// TIA Portal project "Assembler-Analog" (V15.1)

(* hardware
DEVICE "S7-1200 station_1"  S7-1200 Station
   slot 0: "Rack_0"  S7-1200 Rack  Rack  V1.0
   slot 1: "PLC_1"  CPU 1211C DC/DC/DC  6ES7 211-1AE40-0XB0  V4.2
DEVICE "HMI_1"  KTP900 Basic PN
   slot 0: "HMI_1"  KTP900 Basic PN  6AV2 123-2JB03-0AX0  15.1.0.0
   slot 1: "HMI_RT_1"  KTP900 Basic PN  6AV2 123-2JB03-0AX0  15.1.0.0
   slot 5: "HMI_1.IE_CP_1"  PROFINET Interface  15.0.1.0
      slot 1: "PROFINET Interface_1"  PROFINET Interface
         slot 1: "Port_1"  Port
*)

// ===== PLC "PLC_1"  CPU 1211C DC/DC/DC =====

VAR_GLOBAL   // PLC tag table "Default tag table"
   "Clock_Byte" AT %MB1869 : Byte;
   "Clock_10Hz" AT %M1869.0 : Bool;
   "Clock_5Hz" AT %M1869.1 : Bool;
   "Clock_2.5Hz" AT %M1869.2 : Bool;
   "Clock_2Hz" AT %M1869.3 : Bool;
   "Clock_1.25Hz" AT %M1869.4 : Bool;
   "Clock_1Hz" AT %M1869.5 : Bool;
   "Clock_0.625Hz" AT %M1869.6 : Bool;
   "Clock_0.5Hz" AT %M1869.7 : Bool;
   "System_Byte" AT %MB869 : Byte;
   "FirstScan" AT %M869.0 : Bool;
   "DiagStatusUpdate" AT %M869.1 : Bool;
   "AlwaysTRUE" AT %M869.2 : Bool;
   "AlwaysFALSE" AT %M869.3 : Bool;
END_VAR

VAR_GLOBAL   // PLC tag table "aux"
   "counting_step_1" AT %MW50 : Int;
   "6_box_set_count" AT %MW52 : Int;
   "counting_step_2" AT %MW54 : Int;
   "6_box_set_2" AT %MW56 : Int;
   "pallet_entry_bit" AT %M1.0 : Bool;
   "pallet_fed_entry_bit" AT %M0.6 : Bool;
   "pallet_loaded_bit" AT %M1.3 : Bool;
   "box_2_check_bit" AT %M0.4 : Bool;
   "box_1_check_bit" AT %M0.2 : Bool;
   "turn_cycle_on" AT %M0.3 : Bool;
   "push_limit_bit" AT %M0.5 : Bool;
   "plate_limit_bit" AT %M1.1 : Bool;
   "elevator_moving_bit" AT %M1.2 : Bool;
   "pallet_exit_bit" AT %M1.4 : Bool;
   "tag_1" AT %M1.5 : Bool;
   "tag_2" AT %M1.6 : Bool;
   "tag_3" AT %M1.7 : Bool;
   "tag_4" AT %M2.0 : Bool;
   "tag_5" AT %M2.1 : Bool;
   "box_counting_bit" AT %M0.1 : Bool;
   "2_Box_cycle_complete" AT %M0.0 : Bool;
END_VAR

VAR_GLOBAL   // PLC tag table "I/O_factory"
   "pallet_at_entry" AT %I1.7 : Bool;
   "pallet_at_exit" AT %I2.0 : Bool;
   "pallet_loaded" AT %I2.1 : Bool;
   "box_at_entry" AT %I2.2 : Bool;
   "pusher_limit" AT %I2.3 : Bool;
   "plate_limit" AT %I2.4 : Bool;
   "clamped" AT %I2.5 : Bool;
   "elevator_moving" AT %I2.6 : Bool;
   "start" AT %I1.0 : Bool;
   "reset" AT %I1.1 : Bool;
   "stop" AT %I1.2 : Bool;
   "emergency_stop" AT %I1.3 : Bool;
   "auto" AT %I1.4 : Bool;
   "running" AT %I1.5 : Bool;
   "pallet_feeder" AT %Q0.0 : Bool;
   "load_pallet" AT %Q0.1 : Bool;
   "exit_conveyor" AT %Q0.2 : Bool;
   "move_to_limit" AT %Q0.3 : Bool;
   "elevator_up" AT %Q0.4 : Bool;
   "elevator_down" AT %Q0.5 : Bool;
   "box_feeder" AT %Q0.6 : Bool;
   "turn" AT %Q0.7 : Bool;
   "push" AT %Q1.0 : Bool;
   "load_belt" AT %Q1.1 : Bool;
   "clamp" AT %Q1.2 : Bool;
   "open_plate" AT %Q1.3 : Bool;
   "warning_light" AT %Q1.4 : Bool;
   "start_light" AT %Q1.5 : Bool;
   "reset_light" AT %Q1.6 : Bool;
   "stop_light" AT %Q1.7 : Bool;
   "counter" AT %QD30 : DInt;
   "manual" AT %I1.6 : Bool;
END_VAR

DATA_BLOCK "Auxiliare"   // DB1
{ S7_Optimized_Access := 'TRUE' }
VERSION : 0.1
   VAR
      step_counter_1 : Int;
      "6_box_set_count_1" : Int;
      step_count_2 : Int;
      "6_box_set_count_2" : Int;
      "counter" : Int;
      "mod" : DInt;
      turn_cycle_on : Bool;
      system_stop : Bool;
      pallet_entry_elevbit : Bool;
      pallet_fed_entry_bit : Bool;
      pallet_loaded_bit : Bool;
      box2_check_bit : Bool;
      box1_check_bit : Bool;
      "2_box_cycle_complete" : Bool;
      pusher_limit_bit : Bool;
      plate_limit_bit : Bool;
      elevator_moving_bit : Bool;
      pallet_exit_bit : Bool;
      aux1 : Bool;
      aux2 : Bool;
      aux3 : Bool;
      aux4 : Bool;
      aux5 : Bool;
      box_counting_bit : Bool;
   END_VAR
BEGIN
END_DATA_BLOCK

// folder: FBs/Cutii

DATA_BLOCK "Cutii_FB_DB"   // DB5
{ S7_Optimized_Access := 'TRUE' }
VERSION : 0.1
// stored: InstanceOfName Cutii_FB
"Cutii_FB"
BEGIN
END_DATA_BLOCK

// folder: FBs/Paleti

DATA_BLOCK "Paleti_FB_DB"   // DB4
{ S7_Optimized_Access := 'TRUE' }
VERSION : 0.1
// stored: InstanceOfName Paleti_FB
"Paleti_FB"
BEGIN
END_DATA_BLOCK

// folder: FBs/Paletizor

DATA_BLOCK "Paletizor_FB_DB"   // DB2
{ S7_Optimized_Access := 'TRUE' }
VERSION : 0.1
// stored: InstanceOfName Paletizor_FB
"Paletizor_FB"
BEGIN
END_DATA_BLOCK

// folder: System blocks/Program resources

DATA_BLOCK "2_box_timer"   // DB3
{ S7_Optimized_Access := 'TRUE' }
AUTHOR : Simatic
FAMILY : IEC
NAME : IEC_TMR
VERSION : 1.0
// stored: InstanceOfName IEC_TIMER
"IEC_TIMER"
BEGIN
END_DATA_BLOCK

DATA_BLOCK "3_box_timer"   // DB7
{ S7_Optimized_Access := 'TRUE' }
AUTHOR : Simatic
FAMILY : IEC
NAME : IEC_TMR
VERSION : 1.0
// stored: InstanceOfName IEC_TIMER
"IEC_TIMER"
BEGIN
END_DATA_BLOCK

// folder: (top level)

FUNCTION "paletizor" : Void   // FC1, LAD
{ S7_Optimized_Access := 'TRUE' }
VERSION : 0.1
   VAR_TEMP   // added for the SCL form of the ladder/FBD networks
      _w1 : Bool;
      _w2 : Bool;
      _w3 : Bool;
   END_VAR
BEGIN

REGION Network 1: butoane start, stop, reset si esd
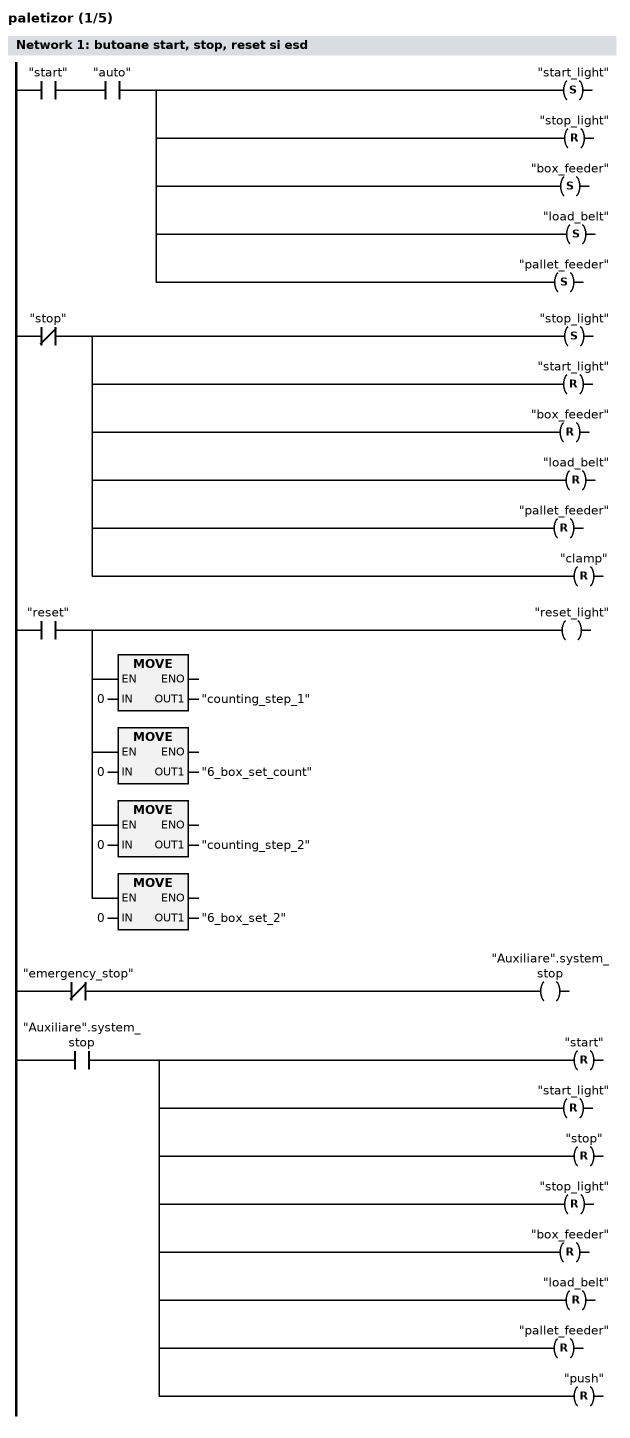
   RUNG wire#powerrail
      Contact( "start" )
      Contact( "auto" )
      wire#w1
      S_Coil( "start_light" )
   END_RUNG
   RUNG wire#w1
      R_Coil( "stop_light" )
   END_RUNG
   RUNG wire#w1
      S_Coil( "box_feeder" )
   END_RUNG
   RUNG wire#w1
      S_Coil( "load_belt" )
   END_RUNG
   RUNG wire#w1
      S_Coil( "pallet_feeder" )
   END_RUNG
   RUNG wire#powerrail
      I_Contact( "stop" )
      wire#w2
      S_Coil( "stop_light" )
   END_RUNG
   RUNG wire#w2
      R_Coil( "start_light" )
   END_RUNG
   RUNG wire#w2
      R_Coil( "box_feeder" )
   END_RUNG
   RUNG wire#w2
      R_Coil( "load_belt" )
   END_RUNG
   RUNG wire#w2
      R_Coil( "pallet_feeder" )
   END_RUNG
   RUNG wire#w2
      R_Coil( "clamp" )
   END_RUNG
   RUNG wire#powerrail
      Contact( "reset" )
      wire#w3
      Coil( "reset_light" )
   END_RUNG
   RUNG wire#w3
      Move(in := 0, out1 => "counting_step_1")
   END_RUNG
   RUNG wire#w3
      Move(in := 0, out1 => "6_box_set_count")
   END_RUNG
   RUNG wire#w3
      Move(in := 0, out1 => "counting_step_2")
   END_RUNG
   RUNG wire#w3
      Move(in := 0, out1 => "6_box_set_2")
   END_RUNG
   RUNG wire#powerrail
      I_Contact( "emergency_stop" )
      Coil( "Auxiliare".system_stop )
   END_RUNG
   RUNG wire#powerrail
      Contact( "Auxiliare".system_stop )
      wire#w4
      R_Coil( "start" )
   END_RUNG
   RUNG wire#w4
      R_Coil( "start_light" )
   END_RUNG
   RUNG wire#w4
      R_Coil( "stop" )
   END_RUNG
   RUNG wire#w4
      R_Coil( "stop_light" )
   END_RUNG
   RUNG wire#w4
      R_Coil( "box_feeder" )
   END_RUNG
   RUNG wire#w4
      R_Coil( "load_belt" )
   END_RUNG
   RUNG wire#w4
      R_Coil( "pallet_feeder" )
   END_RUNG
   RUNG wire#w4
      R_Coil( "push" )
   END_RUNG
   // the same network as SCL:
   IF "start" AND "auto" THEN
       "start_light" := TRUE;
       "stop_light" := FALSE;
       "box_feeder" := TRUE;
       "load_belt" := TRUE;
       "pallet_feeder" := TRUE;
   END_IF;
   IF NOT "stop" THEN
       "stop_light" := TRUE;
       "start_light" := FALSE;
       "box_feeder" := FALSE;
       "load_belt" := FALSE;
       "pallet_feeder" := FALSE;
       "clamp" := FALSE;
   END_IF;
   "reset_light" := "reset";
   IF "reset" THEN
       "counting_step_1" := 0;
       "6_box_set_count" := 0;
       "counting_step_2" := 0;
       "6_box_set_2" := 0;
   END_IF;
   "Auxiliare".system_stop := NOT "emergency_stop";
   IF "Auxiliare".system_stop THEN
       "start" := FALSE;
       "start_light" := FALSE;
       "stop" := FALSE;
       "stop_light" := FALSE;
       "box_feeder" := FALSE;
       "load_belt" := FALSE;
       "pallet_feeder" := FALSE;
       "push" := FALSE;
   END_IF;
END_REGION

REGION Network 2: palet la intrare
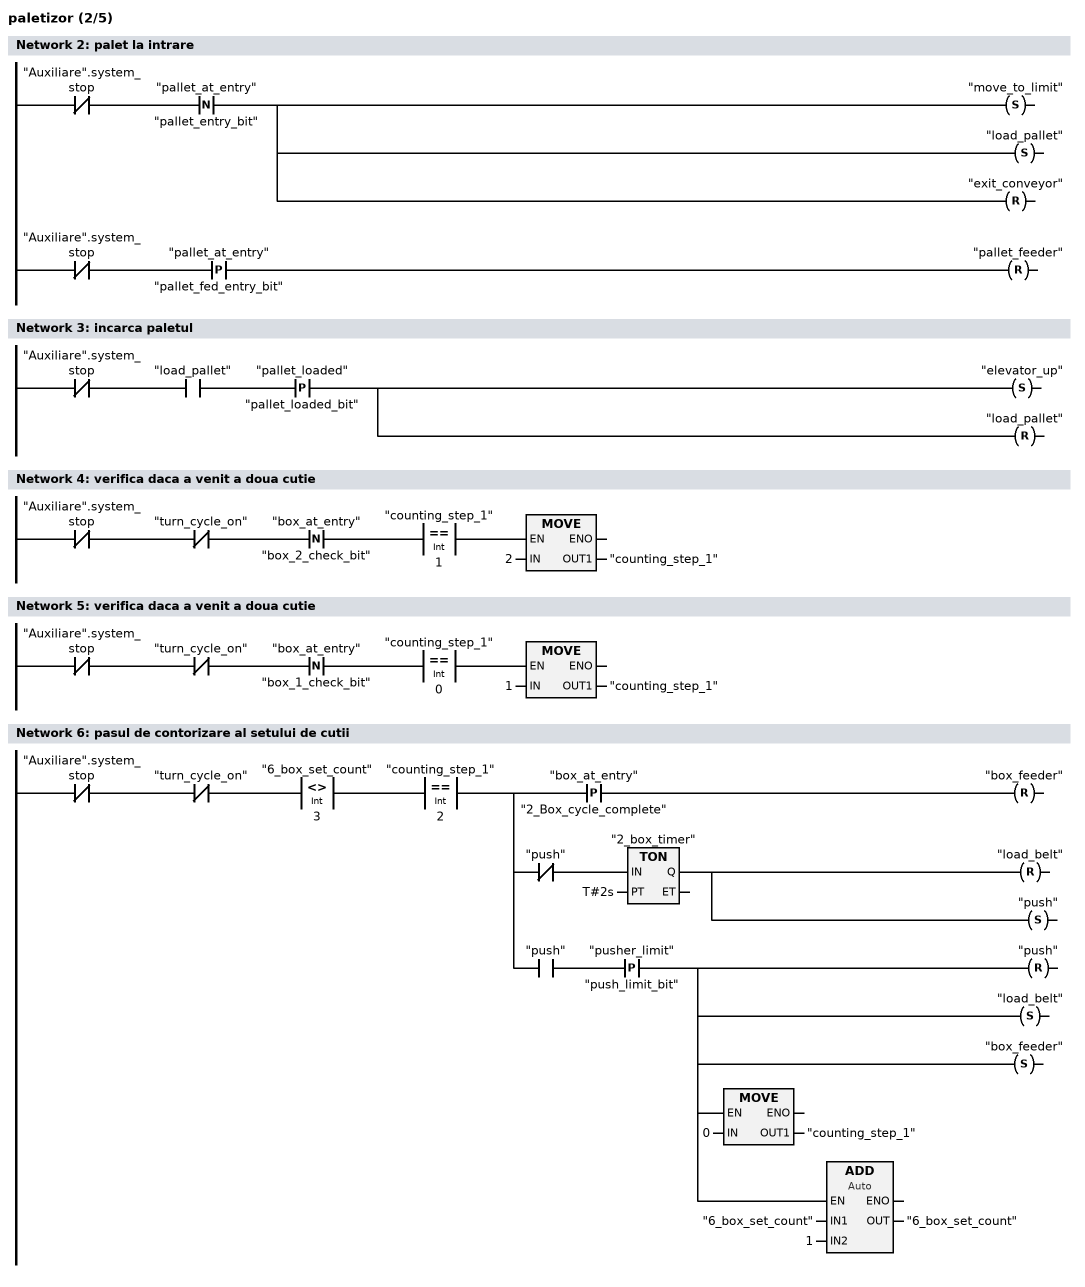
   RUNG wire#powerrail
      I_Contact( "Auxiliare".system_stop )
      N_Contact(operand := "pallet_at_entry", bit := "pallet_entry_bit")
      wire#w1
      S_Coil( "move_to_limit" )
   END_RUNG
   RUNG wire#w1
      S_Coil( "load_pallet" )
   END_RUNG
   RUNG wire#w1
      R_Coil( "exit_conveyor" )
   END_RUNG
   RUNG wire#powerrail
      I_Contact( "Auxiliare".system_stop )
      P_Contact(operand := "pallet_at_entry", bit := "pallet_fed_entry_bit")
      R_Coil( "pallet_feeder" )
   END_RUNG
   // the same network as SCL:
   #_w1 := NOT "Auxiliare".system_stop AND NOT "pallet_at_entry" AND "pallet_entry_bit";   // falling edge of "pallet_at_entry"
   "pallet_entry_bit" := "pallet_at_entry";
   IF #_w1 THEN
       "move_to_limit" := TRUE;
       "load_pallet" := TRUE;
       "exit_conveyor" := FALSE;
   END_IF;
   #_w2 := NOT "Auxiliare".system_stop AND "pallet_at_entry" AND NOT "pallet_fed_entry_bit";   // rising edge of "pallet_at_entry"
   "pallet_fed_entry_bit" := "pallet_at_entry";
   IF #_w2 THEN "pallet_feeder" := FALSE; END_IF;
END_REGION

REGION Network 3: incarca paletul
   RUNG wire#powerrail
      I_Contact( "Auxiliare".system_stop )
      Contact( "load_pallet" )
      P_Contact(operand := "pallet_loaded", bit := "pallet_loaded_bit")
      wire#w1
      S_Coil( "elevator_up" )
   END_RUNG
   RUNG wire#w1
      R_Coil( "load_pallet" )
   END_RUNG
   // the same network as SCL:
   #_w1 := NOT "Auxiliare".system_stop AND "load_pallet" AND "pallet_loaded" AND NOT "pallet_loaded_bit";   // rising edge of "pallet_loaded"
   "pallet_loaded_bit" := "pallet_loaded";
   IF #_w1 THEN
       "elevator_up" := TRUE;
       "load_pallet" := FALSE;
   END_IF;
END_REGION

REGION Network 4: verifica daca a venit a doua cutie
   RUNG wire#powerrail
      I_Contact( "Auxiliare".system_stop )
      I_Contact( "turn_cycle_on" )
      N_Contact(operand := "box_at_entry", bit := "box_2_check_bit")
      { S7_Templates := "SrcType := Int" } EQ_Contact(in1 := "counting_step_1", in2 := 1)
      Move(in := 2, out1 => "counting_step_1")
   END_RUNG
   // the same network as SCL:
   #_w1 := NOT "Auxiliare".system_stop AND NOT "turn_cycle_on" AND NOT "box_at_entry" AND "box_2_check_bit";   // falling edge of "box_at_entry"
   "box_2_check_bit" := "box_at_entry";
   IF #_w1 AND ("counting_step_1" = 1) THEN "counting_step_1" := 2; END_IF;
END_REGION

REGION Network 5: verifica daca a venit a doua cutie
   RUNG wire#powerrail
      I_Contact( "Auxiliare".system_stop )
      I_Contact( "turn_cycle_on" )
      N_Contact(operand := "box_at_entry", bit := "box_1_check_bit")
      { S7_Templates := "SrcType := Int" } EQ_Contact(in1 := "counting_step_1", in2 := 0)
      Move(in := 1, out1 => "counting_step_1")
   END_RUNG
   // the same network as SCL:
   #_w1 := NOT "Auxiliare".system_stop AND NOT "turn_cycle_on" AND NOT "box_at_entry" AND "box_1_check_bit";   // falling edge of "box_at_entry"
   "box_1_check_bit" := "box_at_entry";
   IF #_w1 AND ("counting_step_1" = 0) THEN "counting_step_1" := 1; END_IF;
END_REGION

REGION Network 6: pasul de contorizare al setului de cutii
   #_w1 := NOT "Auxiliare".system_stop AND NOT "turn_cycle_on" AND ("6_box_set_count" <> 3) AND ("counting_step_1" = 2);
   #_w2 := #_w1 AND "box_at_entry" AND NOT "2_Box_cycle_complete";   // rising edge of "box_at_entry"
   "2_Box_cycle_complete" := "box_at_entry";
   IF #_w2 THEN "box_feeder" := FALSE; END_IF;
   "2_box_timer".TON(IN := #_w1 AND NOT "push", PT := T#2s);
   IF "2_box_timer".Q THEN
       "load_belt" := FALSE;
       "push" := TRUE;
   END_IF;
   #_w3 := #_w1 AND "push" AND "pusher_limit" AND NOT "push_limit_bit";   // rising edge of "pusher_limit"
   "push_limit_bit" := "pusher_limit";
   IF #_w3 THEN
       "push" := FALSE;
       "load_belt" := TRUE;
       "box_feeder" := TRUE;
       "counting_step_1" := 0;
       "6_box_set_count" := "6_box_set_count" + 1;
   END_IF;
END_REGION

REGION Network 7: daca s a format setul, sa dea clamp
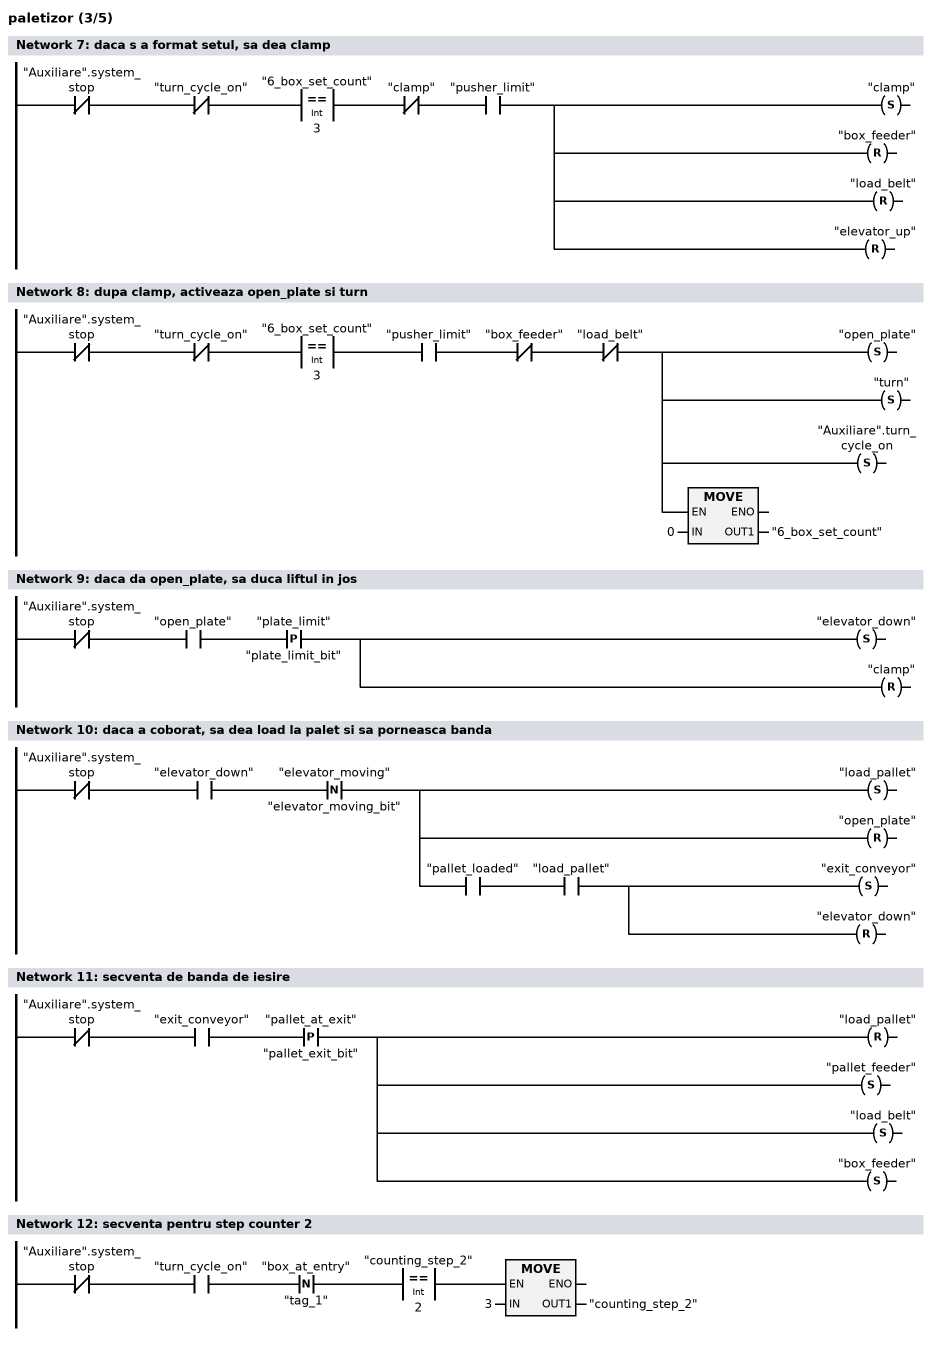
   RUNG wire#powerrail
      I_Contact( "Auxiliare".system_stop )
      I_Contact( "turn_cycle_on" )
      { S7_Templates := "SrcType := Int" } EQ_Contact(in1 := "6_box_set_count", in2 := 3)
      I_Contact( "clamp" )
      Contact( "pusher_limit" )
      wire#w1
      S_Coil( "clamp" )
   END_RUNG
   RUNG wire#w1
      R_Coil( "box_feeder" )
   END_RUNG
   RUNG wire#w1
      R_Coil( "load_belt" )
   END_RUNG
   RUNG wire#w1
      R_Coil( "elevator_up" )
   END_RUNG
   // the same network as SCL:
   #_w1 := NOT "Auxiliare".system_stop AND NOT "turn_cycle_on" AND ("6_box_set_count" = 3) AND NOT "clamp" AND "pusher_limit";
   IF #_w1 THEN
       "clamp" := TRUE;
       "box_feeder" := FALSE;
       "load_belt" := FALSE;
       "elevator_up" := FALSE;
   END_IF;
END_REGION

REGION Network 8: dupa clamp, activeaza open_plate si turn
   RUNG wire#powerrail
      I_Contact( "Auxiliare".system_stop )
      I_Contact( "turn_cycle_on" )
      { S7_Templates := "SrcType := Int" } EQ_Contact(in1 := "6_box_set_count", in2 := 3)
      Contact( "pusher_limit" )
      I_Contact( "box_feeder" )
      I_Contact( "load_belt" )
      wire#w1
      S_Coil( "open_plate" )
   END_RUNG
   RUNG wire#w1
      S_Coil( "turn" )
   END_RUNG
   RUNG wire#w1
      S_Coil( "Auxiliare".turn_cycle_on )
   END_RUNG
   RUNG wire#w1
      Move(in := 0, out1 => "6_box_set_count")
   END_RUNG
   // the same network as SCL:
   IF NOT "Auxiliare".system_stop AND NOT "turn_cycle_on" AND ("6_box_set_count" = 3) AND "pusher_limit" AND NOT "box_feeder" AND NOT "load_belt" THEN
       "open_plate" := TRUE;
       "turn" := TRUE;
       "Auxiliare".turn_cycle_on := TRUE;
       "6_box_set_count" := 0;
   END_IF;
END_REGION

REGION Network 9: daca da open_plate, sa duca liftul in jos
   RUNG wire#powerrail
      I_Contact( "Auxiliare".system_stop )
      Contact( "open_plate" )
      P_Contact(operand := "plate_limit", bit := "plate_limit_bit")
      wire#w1
      S_Coil( "elevator_down" )
   END_RUNG
   RUNG wire#w1
      R_Coil( "clamp" )
   END_RUNG
   // the same network as SCL:
   #_w1 := NOT "Auxiliare".system_stop AND "open_plate" AND "plate_limit" AND NOT "plate_limit_bit";   // rising edge of "plate_limit"
   "plate_limit_bit" := "plate_limit";
   IF #_w1 THEN
       "elevator_down" := TRUE;
       "clamp" := FALSE;
   END_IF;
END_REGION

REGION Network 10: daca a coborat, sa dea load la palet si sa porneasca banda
   RUNG wire#powerrail
      I_Contact( "Auxiliare".system_stop )
      Contact( "elevator_down" )
      N_Contact(operand := "elevator_moving", bit := "elevator_moving_bit")
      wire#w1
      S_Coil( "load_pallet" )
   END_RUNG
   RUNG wire#w1
      R_Coil( "open_plate" )
   END_RUNG
   RUNG wire#w1
      Contact( "pallet_loaded" )
      Contact( "load_pallet" )
      wire#w2
      S_Coil( "exit_conveyor" )
   END_RUNG
   RUNG wire#w2
      R_Coil( "elevator_down" )
   END_RUNG
   // the same network as SCL:
   #_w1 := NOT "Auxiliare".system_stop AND "elevator_down" AND NOT "elevator_moving" AND "elevator_moving_bit";   // falling edge of "elevator_moving"
   "elevator_moving_bit" := "elevator_moving";
   IF #_w1 THEN
       "load_pallet" := TRUE;
       "open_plate" := FALSE;
   END_IF;
   IF #_w1 AND "pallet_loaded" AND "load_pallet" THEN
       "exit_conveyor" := TRUE;
       "elevator_down" := FALSE;
   END_IF;
END_REGION

REGION Network 11: secventa de banda de iesire
   RUNG wire#powerrail
      I_Contact( "Auxiliare".system_stop )
      Contact( "exit_conveyor" )
      P_Contact(operand := "pallet_at_exit", bit := "pallet_exit_bit")
      wire#w1
      R_Coil( "load_pallet" )
   END_RUNG
   RUNG wire#w1
      S_Coil( "pallet_feeder" )
   END_RUNG
   RUNG wire#w1
      S_Coil( "load_belt" )
   END_RUNG
   RUNG wire#w1
      S_Coil( "box_feeder" )
   END_RUNG
   // the same network as SCL:
   #_w1 := NOT "Auxiliare".system_stop AND "exit_conveyor" AND "pallet_at_exit" AND NOT "pallet_exit_bit";   // rising edge of "pallet_at_exit"
   "pallet_exit_bit" := "pallet_at_exit";
   IF #_w1 THEN
       "load_pallet" := FALSE;
       "pallet_feeder" := TRUE;
       "load_belt" := TRUE;
       "box_feeder" := TRUE;
   END_IF;
END_REGION

REGION Network 12: secventa pentru step counter 2
   RUNG wire#powerrail
      I_Contact( "Auxiliare".system_stop )
      Contact( "turn_cycle_on" )
      N_Contact(operand := "box_at_entry", bit := "tag_1")
      { S7_Templates := "SrcType := Int" } EQ_Contact(in1 := "counting_step_2", in2 := 2)
      Move(in := 3, out1 => "counting_step_2")
   END_RUNG
   // the same network as SCL:
   #_w1 := NOT "Auxiliare".system_stop AND "turn_cycle_on" AND NOT "box_at_entry" AND "tag_1";   // falling edge of "box_at_entry"
   "tag_1" := "box_at_entry";
   IF #_w1 AND ("counting_step_2" = 2) THEN "counting_step_2" := 3; END_IF;
END_REGION

REGION Network 13: secventa pentru step counter 2, partea precedenta
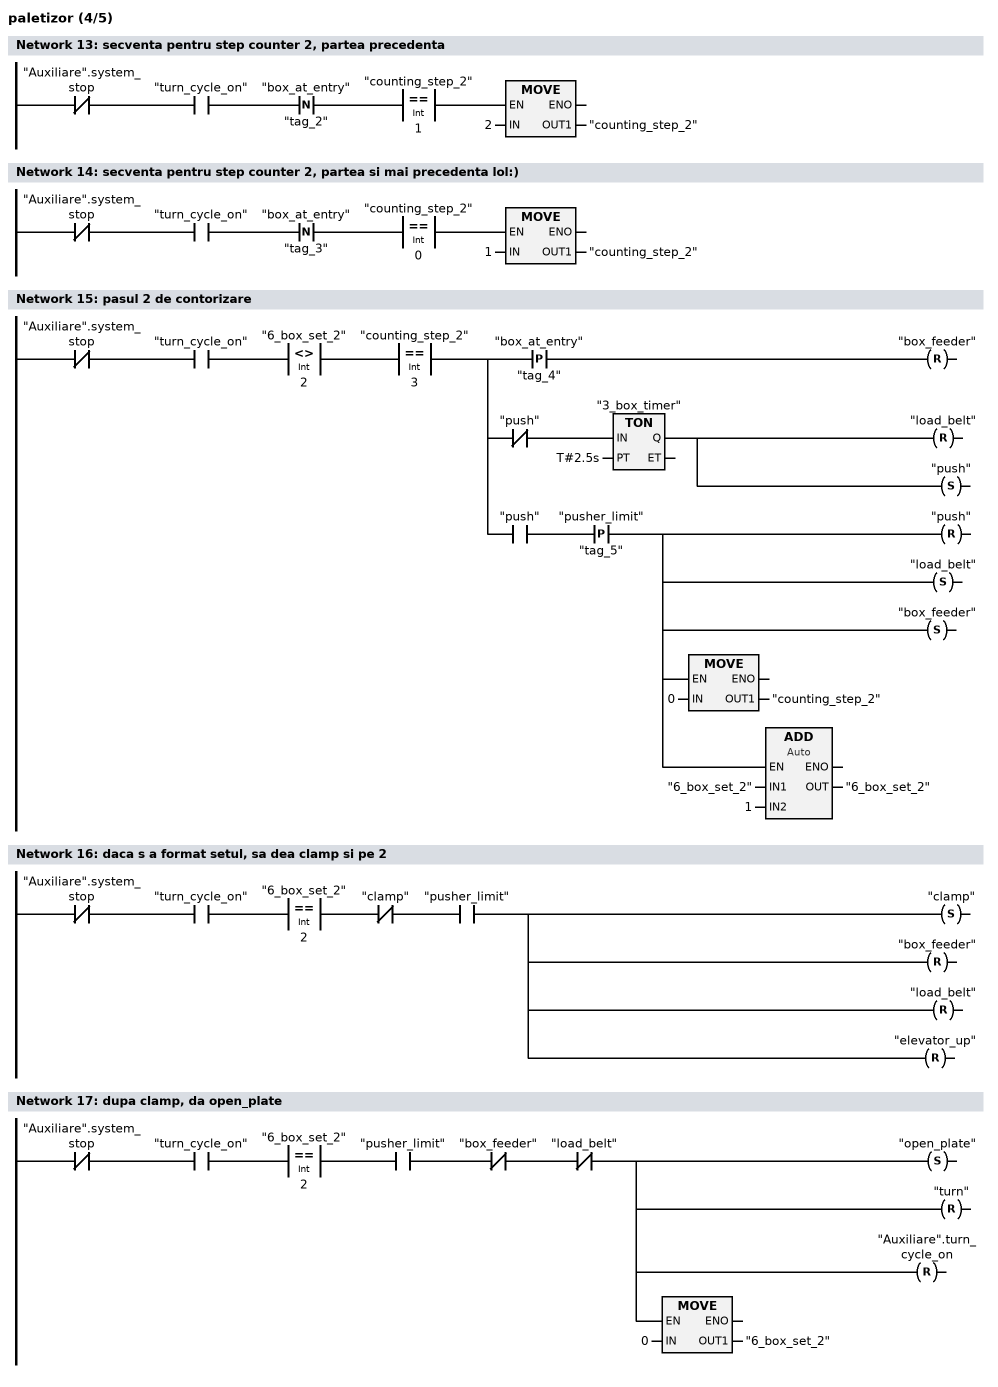
   RUNG wire#powerrail
      I_Contact( "Auxiliare".system_stop )
      Contact( "turn_cycle_on" )
      N_Contact(operand := "box_at_entry", bit := "tag_2")
      { S7_Templates := "SrcType := Int" } EQ_Contact(in1 := "counting_step_2", in2 := 1)
      Move(in := 2, out1 => "counting_step_2")
   END_RUNG
   // the same network as SCL:
   #_w1 := NOT "Auxiliare".system_stop AND "turn_cycle_on" AND NOT "box_at_entry" AND "tag_2";   // falling edge of "box_at_entry"
   "tag_2" := "box_at_entry";
   IF #_w1 AND ("counting_step_2" = 1) THEN "counting_step_2" := 2; END_IF;
END_REGION

REGION Network 14: secventa pentru step counter 2, partea si mai precedenta lol:)
   RUNG wire#powerrail
      I_Contact( "Auxiliare".system_stop )
      Contact( "turn_cycle_on" )
      N_Contact(operand := "box_at_entry", bit := "tag_3")
      { S7_Templates := "SrcType := Int" } EQ_Contact(in1 := "counting_step_2", in2 := 0)
      Move(in := 1, out1 => "counting_step_2")
   END_RUNG
   // the same network as SCL:
   #_w1 := NOT "Auxiliare".system_stop AND "turn_cycle_on" AND NOT "box_at_entry" AND "tag_3";   // falling edge of "box_at_entry"
   "tag_3" := "box_at_entry";
   IF #_w1 AND ("counting_step_2" = 0) THEN "counting_step_2" := 1; END_IF;
END_REGION

REGION Network 15: pasul 2 de contorizare
   #_w1 := NOT "Auxiliare".system_stop AND "turn_cycle_on" AND ("6_box_set_2" <> 2) AND ("counting_step_2" = 3);
   #_w2 := #_w1 AND "box_at_entry" AND NOT "tag_4";   // rising edge of "box_at_entry"
   "tag_4" := "box_at_entry";
   IF #_w2 THEN "box_feeder" := FALSE; END_IF;
   "3_box_timer".TON(IN := #_w1 AND NOT "push", PT := T#2.5s);
   IF "3_box_timer".Q THEN
       "load_belt" := FALSE;
       "push" := TRUE;
   END_IF;
   #_w3 := #_w1 AND "push" AND "pusher_limit" AND NOT "tag_5";   // rising edge of "pusher_limit"
   "tag_5" := "pusher_limit";
   IF #_w3 THEN
       "push" := FALSE;
       "load_belt" := TRUE;
       "box_feeder" := TRUE;
       "counting_step_2" := 0;
       "6_box_set_2" := "6_box_set_2" + 1;
   END_IF;
END_REGION

REGION Network 16: daca s a format setul, sa dea clamp si pe 2
   RUNG wire#powerrail
      I_Contact( "Auxiliare".system_stop )
      Contact( "turn_cycle_on" )
      { S7_Templates := "SrcType := Int" } EQ_Contact(in1 := "6_box_set_2", in2 := 2)
      I_Contact( "clamp" )
      Contact( "pusher_limit" )
      wire#w1
      S_Coil( "clamp" )
   END_RUNG
   RUNG wire#w1
      R_Coil( "box_feeder" )
   END_RUNG
   RUNG wire#w1
      R_Coil( "load_belt" )
   END_RUNG
   RUNG wire#w1
      R_Coil( "elevator_up" )
   END_RUNG
   // the same network as SCL:
   #_w1 := NOT "Auxiliare".system_stop AND "turn_cycle_on" AND ("6_box_set_2" = 2) AND NOT "clamp" AND "pusher_limit";
   IF #_w1 THEN
       "clamp" := TRUE;
       "box_feeder" := FALSE;
       "load_belt" := FALSE;
       "elevator_up" := FALSE;
   END_IF;
END_REGION

REGION Network 17: dupa clamp, da open_plate
   RUNG wire#powerrail
      I_Contact( "Auxiliare".system_stop )
      Contact( "turn_cycle_on" )
      { S7_Templates := "SrcType := Int" } EQ_Contact(in1 := "6_box_set_2", in2 := 2)
      Contact( "pusher_limit" )
      I_Contact( "box_feeder" )
      I_Contact( "load_belt" )
      wire#w1
      S_Coil( "open_plate" )
   END_RUNG
   RUNG wire#w1
      R_Coil( "turn" )
   END_RUNG
   RUNG wire#w1
      R_Coil( "Auxiliare".turn_cycle_on )
   END_RUNG
   RUNG wire#w1
      Move(in := 0, out1 => "6_box_set_2")
   END_RUNG
   // the same network as SCL:
   IF NOT "Auxiliare".system_stop AND "turn_cycle_on" AND ("6_box_set_2" = 2) AND "pusher_limit" AND NOT "box_feeder" AND NOT "load_belt" THEN
       "open_plate" := TRUE;
       "turn" := FALSE;
       "Auxiliare".turn_cycle_on := FALSE;
       "6_box_set_2" := 0;
   END_IF;
END_REGION

REGION Network 18: daca s a terminat, da increment la counter
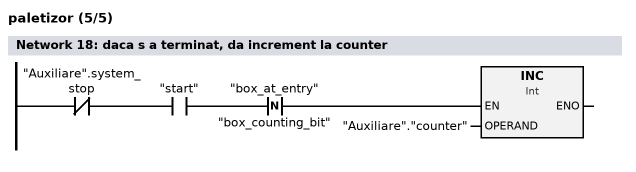
   RUNG wire#powerrail
      I_Contact( "Auxiliare".system_stop )
      Contact( "start" )
      N_Contact(operand := "box_at_entry", bit := "box_counting_bit")
      { S7_Templates := "DestType := Int" } Inc( "Auxiliare"."counter" )
   END_RUNG
   // the same network as SCL:
   #_w1 := NOT "Auxiliare".system_stop AND "start" AND NOT "box_at_entry" AND "box_counting_bit";   // falling edge of "box_at_entry"
   "box_counting_bit" := "box_at_entry";
   IF #_w1 THEN "Auxiliare"."counter" := "Auxiliare"."counter" + 1; END_IF;
END_REGION
END_FUNCTION

FUNCTION "MHJ-PLC-Lab-Function-S71200" : Void   // FC9000, SCL
{ S7_Optimized_Access := 'TRUE' }
VERSION : 0.1
   VAR_TEMP
      rdTimeReturn : Int;
      outputTime : DTL;
      SyncVal : Byte;
      forVal : Int;
      forVal_2 : Int;
      Value : Byte;
   END_VAR
   VAR CONSTANT
      CompVal : Byte := 16#34;
      Value_01 : Byte := 16#11;
      Value_01_DW : DWord := 16#A165_D992;
      Value_02_DW : DWord := 16#58BE_4401;
   END_VAR
BEGIN

   #Value:=PEEK(area := 16#82,
        dbNumber := 0,
        byteOffset := 511);
   #Value := #Value + 1;

   POKE(area := 16#82,
        dbNumber := 0,
        byteOffset := 511,
        value := #Value);

   POKE(area:=16#81,
        dbNumber:=0,
        byteOffset:=1016,
        value:=#Value_01_DW);
   POKE(area := 16#81,
        dbNumber := 0,
        byteOffset := 1020,
        value := #Value_02_DW);

   POKE(area := 16#81,
        dbNumber := 0,
        byteOffset := 511,
        value := B#16#00);

   FOR #forVal := 0 TO 120 DO
       FOR #forVal_2:=0 TO 10 DO
           #rdTimeReturn:=RD_SYS_T(#outputTime);
           #rdTimeReturn := WR_SYS_T(#outputTime);
           #rdTimeReturn := RD_SYS_T(#outputTime);
           #rdTimeReturn := WR_SYS_T(#outputTime);
       END_FOR;
       #SyncVal:= PEEK(area := 16#81,
                      dbNumber := 0,
                      byteOffset := 511);
       IF #SyncVal = #CompVal THEN
          GOTO M_1;
       END_IF;
   END_FOR;
   RETURN;

   M_1:
   POKE(area := 16#81,
        dbNumber := 0,
        byteOffset := 511,
        value := B#16#0);
END_FUNCTION

ORGANIZATION_BLOCK "Main"   // OB1, LAD, ProgramCycle
TITLE = "Main Program Sweep (Cycle)"
{ S7_Optimized_Access := 'TRUE' }
VERSION : 0.1
   VAR_INPUT
      Initial_Call : Bool;   // Initial call of this OB
      Remanence : Bool;   // =True, if remanent data are available
   END_VAR
BEGIN

REGION Network 1: fct de conectare la factory io
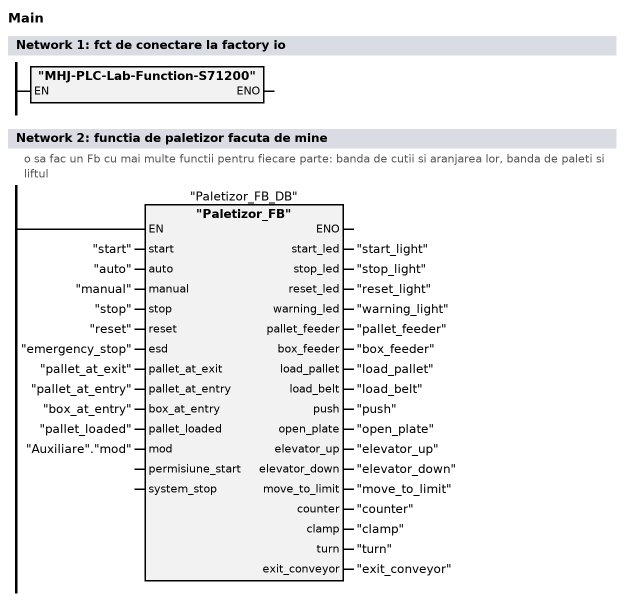
   RUNG wire#powerrail
      "MHJ-PLC-Lab-Function-S71200"()
   END_RUNG
   // the same network as SCL:
   "MHJ-PLC-Lab-Function-S71200"();
END_REGION

REGION Network 2: functia de paletizor facuta de mine
   // o sa fac un Fb cu mai multe functii pentru fiecare parte: banda de cutii si aranjarea lor, banda de paleti si  liftul
   RUNG wire#powerrail
      "Paletizor_FB_DB"(start := "start", auto := "auto", manual := "manual", stop := "stop", reset := "reset", esd := "emergency_stop", pallet_at_exit := "pallet_at_exit", pallet_at_entry := "pallet_at_entry", box_at_entry := "box_at_entry", pallet_loaded := "pallet_loaded", "mod" := "Auxiliare"."mod", permisiune_start :=, system_stop :=, start_led => "start_light", stop_led => "stop_light", reset_led => "reset_light", warning_led => "warning_light", pallet_feeder => "pallet_feeder", box_feeder => "box_feeder", load_pallet => "load_pallet", load_belt => "load_belt", push => "push", open_plate => "open_plate", elevator_up => "elevator_up", elevator_down => "elevator_down", move_to_limit => "move_to_limit", "counter" => "counter", clamp => "clamp", turn => "turn", exit_conveyor => "exit_conveyor")
   END_RUNG
   // the same network as SCL:
   "Paletizor_FB_DB"(start := "start",   // "Paletizor_FB"
                     auto := "auto",
                     manual := "manual",
                     stop := "stop",
                     reset := "reset",
                     esd := "emergency_stop",
                     pallet_at_exit := "pallet_at_exit",
                     pallet_at_entry := "pallet_at_entry",
                     box_at_entry := "box_at_entry",
                     pallet_loaded := "pallet_loaded",
                     "mod" := "Auxiliare"."mod",
                     start_led => "start_light",
                     stop_led => "stop_light",
                     reset_led => "reset_light",
                     warning_led => "warning_light",
                     pallet_feeder => "pallet_feeder",
                     box_feeder => "box_feeder",
                     load_pallet => "load_pallet",
                     load_belt => "load_belt",
                     push => "push",
                     open_plate => "open_plate",
                     elevator_up => "elevator_up",
                     elevator_down => "elevator_down",
                     move_to_limit => "move_to_limit",
                     "counter" => "counter",
                     clamp => "clamp",
                     turn => "turn",
                     exit_conveyor => "exit_conveyor");
END_REGION
END_ORGANIZATION_BLOCK

// folder: FBs/Cutii

FUNCTION_BLOCK "Cutii_FB"   // FB2, LAD
{ S7_Optimized_Access := 'TRUE' }
VERSION : 0.1
   VAR_INPUT
      box_at_entry : Bool;
      permisiune_start : Bool;
      reset : Bool;
      pallet_At_exit : Bool;
      "mod" : DInt;
   END_VAR
   VAR_OUTPUT
      gata_cutii : Bool;
      box_feeder : Bool;
      load_belt : Bool;
      push : Bool;
      clamp : Bool;
      open_plate : Bool;
   END_VAR
   VAR
      counter_box_2 : DInt;
      counter_box_3 : DInt;
      c2_aux : Bool;
      c3_aux : Bool;
      "timer" : TON_TIME;
      timer_1 : TON_TIME;
      timer_2 : TON_TIME;
      timer_3 : TON_TIME;
      timer_4 : TON_TIME;
      timer_5 : TON_TIME;
      timer_gata : Bool;
      timer_gata_1 : Bool;
      aux1 : Bool;
      aux2 : Bool;
      secventa32_gata : Bool;
   END_VAR
   VAR_TEMP   // added for the SCL form of the ladder/FBD networks
      _w1 : Bool;
   END_VAR
BEGIN

REGION Network 1: conditii la cele 2 benzi
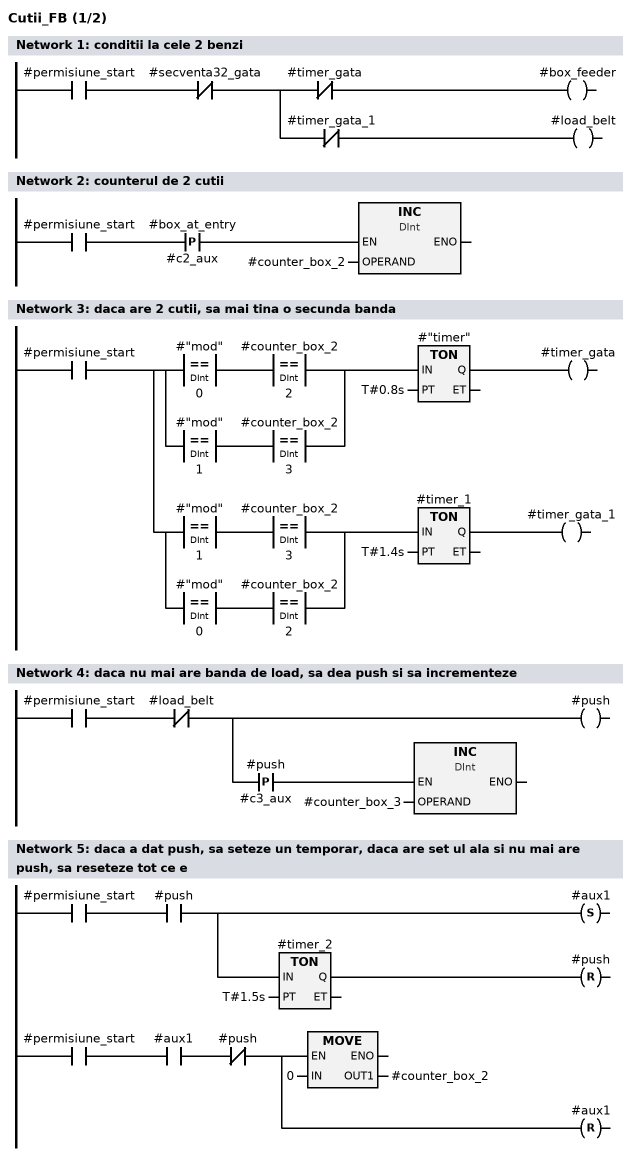
   RUNG wire#powerrail
      Contact( #permisiune_start )
      I_Contact( #secventa32_gata )
      wire#w1
      I_Contact( #timer_gata )
      Coil( #box_feeder )
   END_RUNG
   RUNG wire#w1
      I_Contact( #timer_gata_1 )
      Coil( #load_belt )
   END_RUNG
   // the same network as SCL:
   #_w1 := #permisiune_start AND NOT #secventa32_gata;
   #box_feeder := #_w1 AND NOT #timer_gata;
   #load_belt := #_w1 AND NOT #timer_gata_1;
END_REGION

REGION Network 2: counterul de 2 cutii
   RUNG wire#powerrail
      Contact( #permisiune_start )
      P_Contact(operand := #box_at_entry, bit := #c2_aux)
      { S7_Templates := "DestType := DInt" } Inc( #counter_box_2 )
   END_RUNG
   // the same network as SCL:
   #_w1 := #permisiune_start AND #box_at_entry AND NOT #c2_aux;   // rising edge of #box_at_entry
   #c2_aux := #box_at_entry;
   IF #_w1 THEN #counter_box_2 := #counter_box_2 + 1; END_IF;
END_REGION

REGION Network 3: daca are 2 cutii, sa mai tina o secunda banda
   #"timer"(IN := #permisiune_start AND (((#"mod" = 0) AND (#counter_box_2 = 2)) OR ((#"mod" = 1) AND (#counter_box_2 = 3))),   // TON
            PT := T#0.8s);
   #timer_gata := #"timer".Q;
   #timer_1(IN := #permisiune_start AND (((#"mod" = 1) AND (#counter_box_2 = 3)) OR ((#"mod" = 0) AND (#counter_box_2 = 2))),   // TON
            PT := T#1.4s);
   #timer_gata_1 := #timer_1.Q;
END_REGION

REGION Network 4: daca nu mai are banda de load, sa dea push si sa incrementeze
   RUNG wire#powerrail
      Contact( #permisiune_start )
      I_Contact( #load_belt )
      wire#w1
      Coil( #push )
   END_RUNG
   RUNG wire#w1
      P_Contact(operand := #push, bit := #c3_aux)
      { S7_Templates := "DestType := DInt" } Inc( #counter_box_3 )
   END_RUNG
   // the same network as SCL:
   #push := #permisiune_start AND NOT #load_belt;
   #_w1 := #push AND #push AND NOT #c3_aux;   // rising edge of #push
   #c3_aux := #push;
   IF #_w1 THEN #counter_box_3 := #counter_box_3 + 1; END_IF;
END_REGION

REGION Network 5: daca a dat push, sa seteze un temporar, daca are set ul ala si nu mai are push, sa reseteze tot ce e
   #_w1 := #permisiune_start AND #push;
   IF #_w1 THEN #aux1 := TRUE; END_IF;
   #timer_2(IN := #_w1, PT := T#1.5s);   // TON
   IF #timer_2.Q THEN #push := FALSE; END_IF;
   IF #permisiune_start AND #aux1 AND NOT #push THEN
       #counter_box_2 := 0;
       #aux1 := FALSE;
   END_IF;
END_REGION

REGION Network 6: daca are cele 6 cutii puse, sa dea ca s a terminat secventa
   // dupa incepe clamp, open, elevator, etc
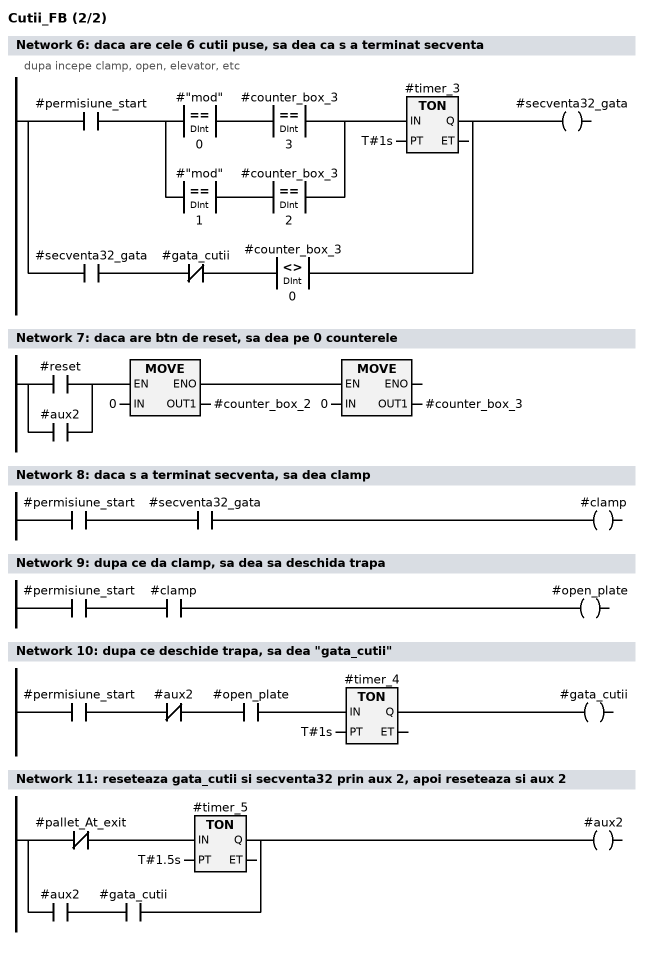
   #timer_3(IN := #permisiune_start AND (((#"mod" = 0) AND (#counter_box_3 = 3)) OR ((#"mod" = 1) AND (#counter_box_3 = 2))),   // TON
            PT := T#1s);
   #secventa32_gata := #timer_3.Q OR (#secventa32_gata AND NOT #gata_cutii AND (#counter_box_3 <> 0));
END_REGION

REGION Network 7: daca are btn de reset, sa dea pe 0 counterele
   RUNG wire#powerrail
      Contact( #reset )
      wire#w1
      Move(in := 0, out1 => #counter_box_2)
      Move(in := 0, out1 => #counter_box_3)
   END_RUNG
   RUNG wire#powerrail
      Contact( #aux2 )
   END_RUNG wire#w1
   // the same network as SCL:
   IF #reset OR #aux2 THEN
       #counter_box_2 := 0;
       #counter_box_3 := 0;
   END_IF;
END_REGION

REGION Network 8: daca s a terminat secventa, sa dea clamp
   RUNG wire#powerrail
      Contact( #permisiune_start )
      Contact( #secventa32_gata )
      Coil( #clamp )
   END_RUNG
   // the same network as SCL:
   #clamp := #permisiune_start AND #secventa32_gata;
END_REGION

REGION Network 9: dupa ce da clamp, sa dea sa deschida trapa
   RUNG wire#powerrail
      Contact( #permisiune_start )
      Contact( #clamp )
      Coil( #open_plate )
   END_RUNG
   // the same network as SCL:
   #open_plate := #permisiune_start AND #clamp;
END_REGION

REGION Network 10: dupa ce deschide trapa, sa dea "gata_cutii"
   #timer_4(IN := #permisiune_start AND NOT #aux2 AND #open_plate, PT := T#1s);   // TON
   #gata_cutii := #timer_4.Q;
END_REGION

REGION Network 11: reseteaza gata_cutii si secventa32 prin aux 2, apoi reseteaza si aux 2
   #timer_5(IN := NOT #pallet_At_exit, PT := T#1.5s);   // TON
   #aux2 := #timer_5.Q OR (#aux2 AND #gata_cutii);
END_REGION
END_FUNCTION_BLOCK

// folder: FBs/Paleti

FUNCTION_BLOCK "Paleti_FB"   // FB3, LAD
{ S7_Optimized_Access := 'TRUE' }
VERSION : 0.1
   VAR_INPUT
      permisiune_Start : Bool;
      pallet_at_entry : Bool;
      pallet_at_exit : Bool;
      pallet_loaded : Bool;
      gata_cutii : Bool;
      open_plate : Bool;
      reset : Bool;
      stop : Bool;
      esd : Bool;
   END_VAR
   VAR_OUTPUT
      load_pallet : Bool;
      pallet_feeder : Bool;
      elevator_up : Bool;
      elevator_down : Bool;
      move_to_limit : Bool;
      exit_conveyor : Bool;
   END_VAR
   VAR
      "timer" : TON_TIME;
      timer_exit : TON_TIME;
      timer_aux : TON_TIME;
      timer_aux_1 : TON_TIME;
      trecut_timer : Bool;
      trecut_timer_Exit : Bool;
      setter_aux : Bool;
      aux1 : Bool;
      aux2 : Bool;
      aux3 : Bool;
      aux4 : Bool;
      aux5 : Bool;
   END_VAR
BEGIN

REGION Network 1: daca are permisiune si nu a trecut timerul, sa i dea pe banda
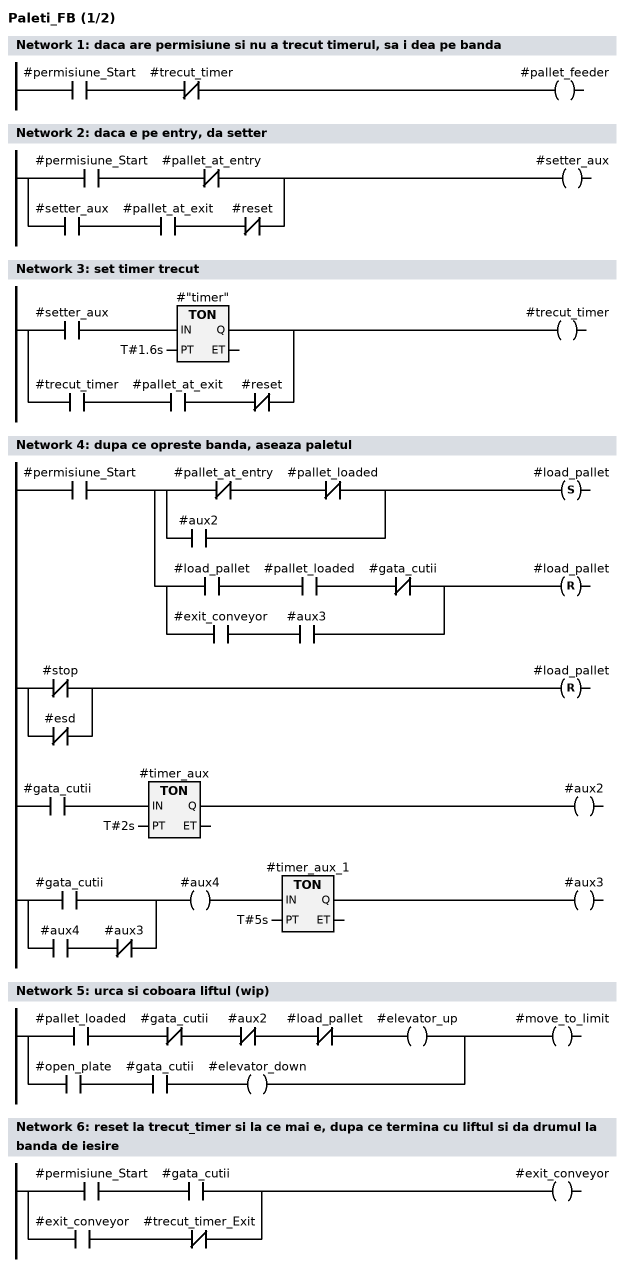
   RUNG wire#powerrail
      Contact( #permisiune_Start )
      I_Contact( #trecut_timer )
      Coil( #pallet_feeder )
   END_RUNG
   // the same network as SCL:
   #pallet_feeder := #permisiune_Start AND NOT #trecut_timer;
END_REGION

REGION Network 2: daca e pe entry, da setter
   RUNG wire#powerrail
      Contact( #permisiune_Start )
      I_Contact( #pallet_at_entry )
      wire#w1
      Coil( #setter_aux )
   END_RUNG
   RUNG wire#powerrail
      Contact( #setter_aux )
      Contact( #pallet_at_exit )
      I_Contact( #reset )
   END_RUNG wire#w1
   // the same network as SCL:
   #setter_aux := (#permisiune_Start AND NOT #pallet_at_entry) OR (#setter_aux AND #pallet_at_exit AND NOT #reset);
END_REGION

REGION Network 3: set timer trecut
   #"timer"(IN := #setter_aux, PT := T#1.6s);   // TON
   #trecut_timer := #"timer".Q OR (#trecut_timer AND #pallet_at_exit AND NOT #reset);
END_REGION

REGION Network 4: dupa ce opreste banda, aseaza paletul
   IF #permisiune_Start AND ((NOT #pallet_at_entry AND NOT #pallet_loaded) OR #aux2) THEN
       #load_pallet := TRUE;
   END_IF;
   IF #permisiune_Start AND ((#load_pallet AND #pallet_loaded AND NOT #gata_cutii) OR (#exit_conveyor AND #aux3)) THEN
       #load_pallet := FALSE;
   END_IF;
   IF NOT #stop OR NOT #esd THEN #load_pallet := FALSE; END_IF;
   #timer_aux(IN := #gata_cutii, PT := T#2s);   // TON
   #aux2 := #timer_aux.Q;
   #aux4 := #gata_cutii OR (#aux4 AND NOT #aux3);
   #timer_aux_1(IN := #aux4, PT := T#5s);   // TON
   #aux3 := #timer_aux_1.Q;
END_REGION

REGION Network 5: urca si coboara liftul (wip)
   RUNG wire#powerrail
      Contact( #pallet_loaded )
      I_Contact( #gata_cutii )
      I_Contact( #aux2 )
      I_Contact( #load_pallet )
      Coil( #elevator_up )
      wire#w1
      Coil( #move_to_limit )
   END_RUNG
   RUNG wire#powerrail
      Contact( #open_plate )
      Contact( #gata_cutii )
      Coil( #elevator_down )
   END_RUNG wire#w1
   // the same network as SCL:
   #elevator_up := #pallet_loaded AND NOT #gata_cutii AND NOT #aux2 AND NOT #load_pallet;
   #elevator_down := #open_plate AND #gata_cutii;
   #move_to_limit := #elevator_up OR #elevator_down;
END_REGION

REGION Network 6: reset la trecut_timer si la ce mai e, dupa ce termina cu liftul si da drumul la banda de iesire
   RUNG wire#powerrail
      Contact( #permisiune_Start )
      Contact( #gata_cutii )
      wire#w1
      Coil( #exit_conveyor )
   END_RUNG
   RUNG wire#powerrail
      Contact( #exit_conveyor )
      I_Contact( #trecut_timer_Exit )
   END_RUNG wire#w1
   // the same network as SCL:
   #exit_conveyor := (#permisiune_Start AND #gata_cutii) OR (#exit_conveyor AND NOT #trecut_timer_Exit);
END_REGION

REGION Network 7: timer pt exit
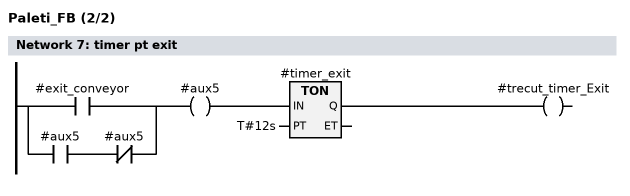
   #aux5 := #exit_conveyor OR (#aux5 AND NOT #aux5);
   #timer_exit(IN := #aux5, PT := T#12s);   // TON
   #trecut_timer_Exit := #timer_exit.Q;
END_REGION
END_FUNCTION_BLOCK

// folder: FBs/Paletizor

FUNCTION_BLOCK "Paletizor_FB"   // FB1, LAD
{ S7_Optimized_Access := 'TRUE' }
VERSION : 0.1
   VAR_INPUT
      start : Bool;
      auto : Bool;
      manual : Bool;
      stop : Bool;
      reset : Bool;
      esd : Bool;
      pallet_at_exit : Bool;
      pallet_at_entry : Bool;
      box_at_entry : Bool;
      pallet_loaded : Bool;
   END_VAR
   VAR_OUTPUT
      start_led : Bool;
      stop_led : Bool;
      reset_led : Bool;
      warning_led : Bool;
      pallet_feeder : Bool;
      box_feeder : Bool;
      load_pallet : Bool;
      load_belt : Bool;
      push : Bool;
      open_plate : Bool;
      elevator_up : Bool;
      elevator_down : Bool;
      move_to_limit : Bool;
      "counter" : DInt;
      clamp : Bool;
      turn : Bool;
      exit_conveyor : Bool;
   END_VAR
   VAR_IN_OUT
      "mod" : DInt;
      permisiune_start : Bool;
      system_stop : Bool;
   END_VAR
   VAR
      gata_cutii : Bool;
      aux_cutii : Bool;
   END_VAR
   VAR_TEMP   // added for the SCL form of the ladder/FBD networks
      _w1 : Bool;
   END_VAR
BEGIN

REGION Network 1: daca e pe start is pe auto, sa dea permisiunea de start
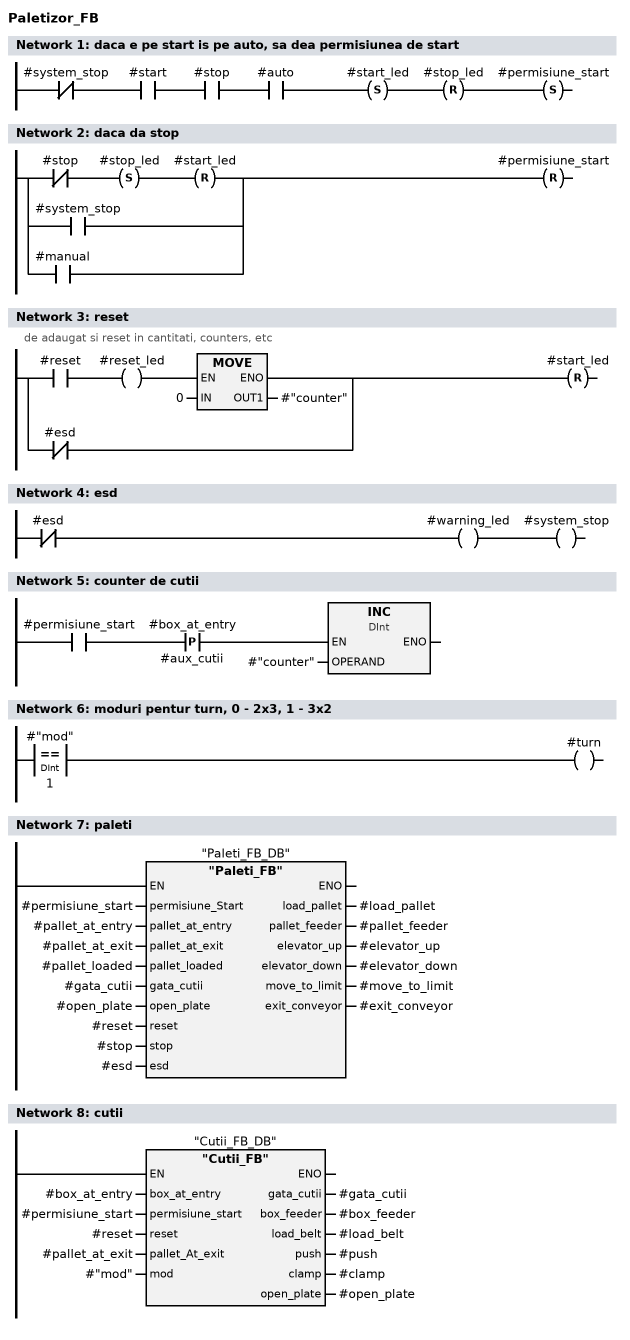
   RUNG wire#powerrail
      I_Contact( #system_stop )
      Contact( #start )
      Contact( #stop )
      Contact( #auto )
      S_Coil( #start_led )
      R_Coil( #stop_led )
      S_Coil( #permisiune_start )
   END_RUNG
   // the same network as SCL:
   IF NOT #system_stop AND #start AND #stop AND #auto THEN
       #start_led := TRUE;
       #stop_led := FALSE;
       #permisiune_start := TRUE;
   END_IF;
END_REGION

REGION Network 2: daca da stop
   RUNG wire#powerrail
      I_Contact( #stop )
      S_Coil( #stop_led )
      R_Coil( #start_led )
      wire#w1
      R_Coil( #permisiune_start )
   END_RUNG
   RUNG wire#powerrail
      Contact( #system_stop )
   END_RUNG wire#w1
   RUNG wire#powerrail
      Contact( #manual )
   END_RUNG wire#w1
   // the same network as SCL:
   IF NOT #stop THEN
       #stop_led := TRUE;
       #start_led := FALSE;
   END_IF;
   IF NOT #stop OR #system_stop OR #manual THEN #permisiune_start := FALSE; END_IF;
END_REGION

REGION Network 3: reset
   // de adaugat si reset in cantitati, counters, etc
   RUNG wire#powerrail
      Contact( #reset )
      Coil( #reset_led )
      Move(in := 0, out1 => #"counter")
      wire#w1
      R_Coil( #start_led )
   END_RUNG
   RUNG wire#powerrail
      I_Contact( #esd )
   END_RUNG wire#w1
   // the same network as SCL:
   #reset_led := #reset;
   IF #reset THEN #"counter" := 0; END_IF;
   IF #reset OR NOT #esd THEN #start_led := FALSE; END_IF;
END_REGION

REGION Network 4: esd
   RUNG wire#powerrail
      I_Contact( #esd )
      Coil( #warning_led )
      Coil( #system_stop )
   END_RUNG
   // the same network as SCL:
   #warning_led := NOT #esd;
   #system_stop := NOT #esd;
END_REGION

REGION Network 5: counter de cutii
   RUNG wire#powerrail
      Contact( #permisiune_start )
      P_Contact(operand := #box_at_entry, bit := #aux_cutii)
      { S7_Templates := "DestType := DInt" } Inc( #"counter" )
   END_RUNG
   // the same network as SCL:
   #_w1 := #permisiune_start AND #box_at_entry AND NOT #aux_cutii;   // rising edge of #box_at_entry
   #aux_cutii := #box_at_entry;
   IF #_w1 THEN #"counter" := #"counter" + 1; END_IF;
END_REGION

REGION Network 6: moduri pentur turn, 0 - 2x3, 1 - 3x2
   RUNG wire#powerrail
      { S7_Templates := "SrcType := DInt" } EQ_Contact(in1 := #"mod", in2 := 1)
      Coil( #turn )
   END_RUNG
   // the same network as SCL:
   #turn := #"mod" = 1;
END_REGION

REGION Network 7: paleti
   RUNG wire#powerrail
      "Paleti_FB_DB"(permisiune_Start := #permisiune_start, pallet_at_entry := #pallet_at_entry, pallet_at_exit := #pallet_at_exit, pallet_loaded := #pallet_loaded, gata_cutii := #gata_cutii, open_plate := #open_plate, reset := #reset, stop := #stop, esd := #esd, load_pallet => #load_pallet, pallet_feeder => #pallet_feeder, elevator_up => #elevator_up, elevator_down => #elevator_down, move_to_limit => #move_to_limit, exit_conveyor => #exit_conveyor)
   END_RUNG
   // the same network as SCL:
   "Paleti_FB_DB"(permisiune_Start := #permisiune_start,   // "Paleti_FB"
                  pallet_at_entry := #pallet_at_entry,
                  pallet_at_exit := #pallet_at_exit,
                  pallet_loaded := #pallet_loaded,
                  gata_cutii := #gata_cutii,
                  open_plate := #open_plate,
                  reset := #reset,
                  stop := #stop,
                  esd := #esd,
                  load_pallet => #load_pallet,
                  pallet_feeder => #pallet_feeder,
                  elevator_up => #elevator_up,
                  elevator_down => #elevator_down,
                  move_to_limit => #move_to_limit,
                  exit_conveyor => #exit_conveyor);
END_REGION

REGION Network 8: cutii
   RUNG wire#powerrail
      "Cutii_FB_DB"(box_at_entry := #box_at_entry, permisiune_start := #permisiune_start, reset := #reset, pallet_At_exit := #pallet_at_exit, "mod" := #"mod", gata_cutii => #gata_cutii, box_feeder => #box_feeder, load_belt => #load_belt, push => #push, clamp => #clamp, open_plate => #open_plate)
   END_RUNG
   // the same network as SCL:
   "Cutii_FB_DB"(box_at_entry := #box_at_entry,   // "Cutii_FB"
                 permisiune_start := #permisiune_start,
                 reset := #reset,
                 pallet_At_exit := #pallet_at_exit,
                 "mod" := #"mod",
                 gata_cutii => #gata_cutii,
                 box_feeder => #box_feeder,
                 load_belt => #load_belt,
                 push => #push,
                 clamp => #clamp,
                 open_plate => #open_plate);
END_REGION
END_FUNCTION_BLOCK

(* ===== HMI "HMI_RT_1" =====
system functions are stored by id; their names below are inferred from use
connection "HMI_Connection_1": ETHERNET, SMART_S7_1200_OMS

HMI tags "Default tag table"
   "counter" : DInt = PLC counter AT %QD30, 1 s
   "Auxiliare_counter" : Int = PLC Auxiliare.counter, 1 s
   "stop_light" : Bool = PLC stop_light AT %Q1.7, 1 s
   "Auxiliare_mod" : DInt = PLC Auxiliare.mod, 1 s
   "start_light" : Bool = PLC start_light AT %Q1.5, 1 s

discrete alarms
   1: 'ESD', class Errors, trigger "Alarme_gather" bit 0

Template "Template_1" 800x480
   Button "Exit" at 722,440 size 55x39; TextOff 'Exit'; PictureOff "ExitRuntime_KTP900_Basic_PN_TR"; PictureOn "ExitRuntime_KTP900_Basic_PN_TR"
      on Release: StopRuntime(0)
   Button "Template_Button" at 622,440 size 55x39; TextOff 'Text'
   Button "Template_Button_1" at 522,440 size 55x39; TextOff 'Text'
   Button "Template_Button_2" at 422,440 size 55x39; TextOff 'Text'
   Button "Template_Button_3" at 322,440 size 55x39; TextOff 'Text'
   Button "Template_Button_4" at 222,440 size 55x39; TextOff 'Text'
   Button "Template_Button_5" at 122,440 size 55x39; TextOff 'Text'
   Button "Template_Button_6" at 22,440 size 55x39; TextOff 'Text'

screen "Main" 800x480, template "Template_1"
   TextField "Text field_1" at 185,103 size 438x25; Text 'Modul poate fi setat doar daca masinaria e pe stop'
   Button "Button_1" at 254,166 size 116x49; TextOff '2x3'
      on Press: SetTag("Auxiliare_mod", 0)
      Visibility <- "start_light"
   Button "Button_2" at 418,165 size 116x49; TextOff '3x2'
      on Press: SetTag("Auxiliare_mod", 1)
      Visibility <- "start_light"
   TextField "Text field_2" at 322,268 size 145x25; Text 'Mod curent: 2x3'
      Visibility <- "Auxiliare_mod"
   TextField "Text field_3" at 322,268 size 145x25; Text 'Mod curent: 3x2'
      Visibility <- "Auxiliare_mod"
*)